# EPICS autosave request: iocBoot/gmca_23b_ioc1/dbSave/digital_IO_24_desc.req
%
% This request file stores settings for PMAC digital out
%

$(P)0.DESC
$(P)1.DESC
$(P)2.DESC
$(P)3.DESC
$(P)4.DESC
$(P)5.DESC
$(P)6.DESC
$(P)7.DESC
$(P)8.DESC
$(P)9.DESC
$(P)10.DESC
$(P)11.DESC
$(P)12.DESC
$(P)13.DESC
$(P)14.DESC
$(P)15.DESC
$(P)16.DESC
$(P)17.DESC
$(P)18.DESC
$(P)19.DESC
$(P)20.DESC
$(P)21.DESC
$(P)22.DESC
$(P)23.DESC
